// TwinCAT 3 PLC project JSON_Luchtvochtigheid
// ProgramVersion: 3.1.4023.0
// libraries:
//   Tc2_Standard, * (Beckhoff Automation GmbH)
//   Tc2_System, * (Beckhoff Automation GmbH)
//   Tc3_IotBase, * (Beckhoff Automation GmbH)
//   Tc3_JsonXml, * (Beckhoff Automation GmbH)
//   Tc3_Module, * (Beckhoff Automation GmbH)
// project tree:
//   / PlcTask.TcTTO
//   POUs/ MAIN.TcPOU
// (motion and I/O tree: see PLC project ftp)
// real-time tasks:
//   TASK PlcTask: cycle T#10ms, priority 20, ADS port 350
//   TASK PlcTask1: cycle T#10ms, priority 21, ADS port 351
//   TASK PlcTask2: cycle T#10ms, priority 22, ADS port 352
//   TASK PlcTask3: cycle T#10ms, priority 23, ADS port 353
//   TASK PlcTask4: cycle T#10ms, priority 24, ADS port 354
//   TASK PlcTask5: cycle T#10ms, priority 25, ADS port 355
//   TASK PlcTask6: cycle T#10ms, priority 26, ADS port 356

CONFIGURATION JSON_Luchtvochtigheid
    RESOURCE PLC ON TwinCAT3
        TASK PlcTask(INTERVAL := T#10ms, PRIORITY := 24);
        PROGRAM MAIN WITH PlcTask : MAIN;
    END_RESOURCE
END_CONFIGURATION

// ---- POUs/MAIN.TcPOU
PROGRAM MAIN
VAR
    // trigger command execution for OpenWeatherMap samples
    bGetOpenWeatherMap: BOOL;	
	bGetContentResult: BOOL;
	
	sContent : STRING(511);
	
	eRequestType: STRING(INT#4);
	RisingEdge: R_TRIG;
	
	FB_IotHttpRequest: FB_IotHttpRequest;
	FB_IotHttpClient: FB_IotHttpClient :=(sHostName := 'observations.buienradar.nl', bKeepAlive := TRUE, tConnectionTimeout := T#10S);
END_VAR

VAR_OUTPUT
	jsonDoc: SJsonValue;
	jsonSerial: SJsonValue;
	fbJson: FB_JsonDomParser;
	humidity : LREAL;
END_VAR

IF NOT FB_IotHttpClient.bConfigured THEN 
    FB_IotHttpClient.stTLS.sCA:= 'C:\Users\Kasper\Desktop\2.cer';
    FB_IotHttpClient.nHostPort:= 443;
    FB_IotHttpClient.stTLS.bNoServerCertCheck:= TRUE;
	
ELSIF FB_IotHttpClient.bConfigured THEN
	bGetOpenWeatherMap := TRUE;
END_IF

RisingEdge(CLK:= bGetOpenWeatherMap);

IF RisingEdge.Q THEN
	IF FB_IotHttpRequest.SendRequest(sUri := '/1.0/actual/weatherstation/10006458?btc=202005061725&ak=66a3435a3dee4dd8b1e8351270ad40fc', fbClient := FB_IotHttpClient, eRequestType := ETcIotHttpRequestType.HTTP_Get, 0, 0, 0) THEN
		bGetContentResult:= FB_IotHttpRequest.GetContent(pContent:= ADR(sContent), nContentSize:= SIZEOF(sContent), bSetNullTermination:= TRUE);
	END_IF
END_IF

IF NOT(FB_IotHttpRequest.bBusy) THEN
	jsonDoc := FB_IotHttpRequest.GetJsonDomContent(fbJson);
	jsonSerial := fbJson.FindMember(jsonDoc, 'humidity');
	humidity := fbJson.GetDouble(jsonSerial);
END_IF

FB_IotHttpClient.Execute();

END_PROGRAM
